TYPE U_AXIS_GEAR_IN :
UNION

  stCtrl              : ARRAY[1..MAX_AXIS] OF ST_GEAR_IN;

  byCtrl    AT %Q*    : ARRAY[1..MAX_AXIS] OF
                        ARRAY[1..SIZEOF(ST_GEAR_IN)] OF BYTE;
END_UNION
END_TYPE

(* stored: Version 1.1.0.1
   DUT U_AXIS_GEAR_IN: Id {cb579414-381f-4b12-ab4c-f0c6501b5f4b} *)
